FUNCTION_BLOCK encodeIOpCdt (* CAT Function Block Type *)
  (* Standard: 61499-2 *)
  (* Version 0.0, 6/7/2026, Schneider Electric, template *)
  PACKAGE SE.Nereda;
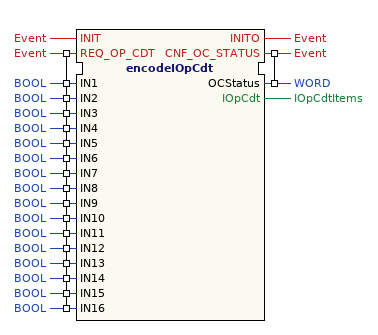
  EVENT_INPUT
    INIT;
    REQ_OP_CDT WITH IN1, IN2, IN3, IN4, IN5, IN6, IN7, IN8, IN9, IN10, IN11, IN12, IN13, IN14, IN15, IN16; (* Normal Execution Request *)
  END_EVENT
  EVENT_OUTPUT
    INITO;
    CNF_OC_STATUS WITH OCStatus; (* Execution Confirmation *)
  END_EVENT
  VAR_INPUT
    IN1 : BOOL; (* Argument *)
    IN2 : BOOL; (* Argument *)
    IN3 : BOOL; (* Argument *)
    IN4 : BOOL; (* Argument *)
    IN5 : BOOL; (* Argument *)
    IN6 : BOOL; (* Argument *)
    IN7 : BOOL; (* Argument *)
    IN8 : BOOL; (* Argument *)
    IN9 : BOOL; (* Argument *)
    IN10 : BOOL; (* Argument *)
    IN11 : BOOL; (* Argument *)
    IN12 : BOOL; (* Argument *)
    IN13 : BOOL; (* Argument *)
    IN14 : BOOL; (* Argument *)
    IN15 : BOOL; (* Argument *)
    IN16 : BOOL; (* Argument *)
  END_VAR
  VAR_OUTPUT
    OCStatus : WORD; (* Output bit image, bit 0 is the LSB of OUT1 *)
  END_VAR
  PLUGS
    IOpCdt : IOpCdtItems;
  END_PLUGS
  (* 01 - FUNCTIONNAL INPUT INTERFACE *)
  (* 05 - LOGIC *)
  (* 02 - FUNCTIONNAL OUTPUT INTERFACE *)
  (* 00 - INITIALIZATION *)
  (* 06 - HMI INTERFACE *)
  (* 03 - FIELD INTERFACE *)
  FBS
    OpCdts : AND_173860434676319F4; {SET_ATTRIBUTE(Configuration.GenericFBType.InterfaceParams, Runtime.Standard#CNT:=16;OUT:BOOL)}
    encodeB1 : VALFORMAT_95B1C22C7F49B890(FORMAT := '%s%s%s%s'); {SET_ATTRIBUTE(Configuration.GenericFBType.InterfaceParams, Runtime.Standard#I:=4;VALUE${I$}:INT,INT,INT,INT)}
    encodeB2 : VALFORMAT_95B1C22C7F49B890(FORMAT := '%s%s%s%s'); {SET_ATTRIBUTE(Configuration.GenericFBType.InterfaceParams, Runtime.Standard#I:=4;VALUE${I$}:INT,INT,INT,INT)}
    OpCdtsSmooth : boolValueChanged;
    encodeB3 : VALFORMAT_95B1C22C7F49B890(FORMAT := '%s%s%s%s'); {SET_ATTRIBUTE(Configuration.GenericFBType.InterfaceParams, Runtime.Standard#I:=4;VALUE${I$}:INT,INT,INT,INT)}
    encodeB4 : VALFORMAT_95B1C22C7F49B890(FORMAT := '%s%s%s%s'); {SET_ATTRIBUTE(Configuration.GenericFBType.InterfaceParams, Runtime.Standard#I:=4;VALUE${I$}:INT,INT,INT,INT)}
    IThis : encodeIOpCdt_HMI(QI := TRUE);
    OC_StatusWordConvert : BITMAN_182F748F2FAD4D59; {SET_ATTRIBUTE(Configuration.GenericFBType.InterfaceParams, Runtime.Standard#CNTIN:=16;CNTOUT:=1;IN${CNTIN$}:BOOL,BOOL,BOOL,BOOL,BOOL,BOOL,BOOL,BOOL,BOOL,BOOL,BOOL,BOOL,BOOL,BOOL,BOOL,BOOL;OUT${CNTOUT$}:WORD)}
    NOT_INs : NOT_21661D42DA8232174; {SET_ATTRIBUTE(Configuration.GenericFBType.InterfaceParams, Runtime.Standard#CNT:=16;OUT${CNT$}:BOOL,BOOL,BOOL,BOOL,BOOL,BOOL,BOOL,BOOL,BOOL,BOOL,BOOL,BOOL,BOOL,BOOL,BOOL,BOOL)}
    STR2INT1 : STR2INT;
    STR2INT2 : STR2INT;
    STR2INT3 : STR2INT;
    STR2INT4 : STR2INT;
    BOOL2INT1 : BOOL2INT_4;
    BOOL2INT2 : BOOL2INT_4;
    BOOL2INT3 : BOOL2INT_4;
    BOOL2INT4 : BOOL2INT_4;
    MemoOCStatus : MemoOC;
    StatusSmooth : WordValueChanged;
  END_FBS
  EVENT_CONNECTIONS
    REQ_OP_CDT TO OpCdts.REQ;
    OpCdts.CNF TO OpCdtsSmooth.REQ;
    OC_StatusWordConvert.INITO TO INITO;
    NOT_INs.CNF TO OC_StatusWordConvert.REQ;
    StatusSmooth.350834820611931F TO CNF_OC_STATUS;
    BOOL2INT1.6FC99A5BD1C38561 TO encodeB1.REQ;
    encodeB1.CNF TO STR2INT1.DD5870AA881150BB;
    BOOL2INT2.6FC99A5BD1C38561 TO encodeB2.REQ;
    encodeB2.CNF TO STR2INT2.DD5870AA881150BB;
    STR2INT1.6FC99A5BD1C38561 TO BOOL2INT2.DD5870AA881150BB;
    BOOL2INT3.6FC99A5BD1C38561 TO encodeB3.REQ;
    encodeB3.CNF TO STR2INT3.DD5870AA881150BB;
    BOOL2INT4.6FC99A5BD1C38561 TO encodeB4.REQ;
    encodeB4.CNF TO STR2INT4.DD5870AA881150BB;
    OpCdtsSmooth.CNF TO BOOL2INT1.DD5870AA881150BB;
    STR2INT2.6FC99A5BD1C38561 TO BOOL2INT3.DD5870AA881150BB;
    STR2INT3.6FC99A5BD1C38561 TO BOOL2INT4.DD5870AA881150BB;
    STR2INT4.6FC99A5BD1C38561 TO NOT_INs.REQ;
    StatusSmooth.350834820611931F TO IOpCdt.0DE1D11A791E8338;
    OpCdtsSmooth.CHD TO IOpCdt.51FD4CCF54DA16B0;
    OC_StatusWordConvert.CNF TO StatusSmooth.77F8F9CFF707DAFF;
    StatusSmooth.93AE3729A9342678 TO MemoOCStatus.7DC0949B91268FF6;
    INIT TO IThis.7D98611DC811A4F7;
    IThis.8A8403C8DB481D6C TO IThis.A665539B906F6DBA;
    MemoOCStatus.3B88FC64E51ED000 TO IThis.E03002787A644D63;
    IThis.8A8403C8DB481D6C TO OC_StatusWordConvert.INIT;
    IThis.6D29BCFC45D76FE3 TO IOpCdt.0DE1D11A791E8338;
    MemoOCStatus.3B88FC64E51ED000 TO IOpCdt.510B9224626AA5DB;
  END_CONNECTIONS
  DATA_CONNECTIONS
    IN1 TO OpCdts.IN1;
    IN2 TO OpCdts.IN2;
    IN16 TO OpCdts.IN16;
    IN15 TO OpCdts.IN15;
    IN14 TO OpCdts.IN14;
    IN13 TO OpCdts.IN13;
    IN12 TO OpCdts.IN12;
    IN11 TO OpCdts.IN11;
    IN10 TO OpCdts.IN10;
    IN9 TO OpCdts.IN9;
    IN8 TO OpCdts.IN8;
    IN7 TO OpCdts.IN7;
    IN6 TO OpCdts.IN6;
    IN5 TO OpCdts.IN5;
    IN4 TO OpCdts.IN4;
    IN3 TO OpCdts.IN3;
    OpCdts.OUT TO OpCdtsSmooth.Input;
    NOT_INs.OUT16 TO OC_StatusWordConvert.IN16;
    NOT_INs.OUT1 TO OC_StatusWordConvert.IN1;
    NOT_INs.OUT2 TO OC_StatusWordConvert.IN2;
    NOT_INs.OUT3 TO OC_StatusWordConvert.IN3;
    NOT_INs.OUT4 TO OC_StatusWordConvert.IN4;
    NOT_INs.OUT5 TO OC_StatusWordConvert.IN5;
    NOT_INs.OUT6 TO OC_StatusWordConvert.IN6;
    NOT_INs.OUT7 TO OC_StatusWordConvert.IN7;
    NOT_INs.OUT8 TO OC_StatusWordConvert.IN8;
    NOT_INs.OUT9 TO OC_StatusWordConvert.IN9;
    NOT_INs.OUT10 TO OC_StatusWordConvert.IN10;
    NOT_INs.OUT11 TO OC_StatusWordConvert.IN11;
    NOT_INs.OUT12 TO OC_StatusWordConvert.IN12;
    NOT_INs.OUT13 TO OC_StatusWordConvert.IN13;
    NOT_INs.OUT14 TO OC_StatusWordConvert.IN14;
    NOT_INs.OUT15 TO OC_StatusWordConvert.IN15;
    IN1 TO NOT_INs.IN1;
    IN2 TO NOT_INs.IN2;
    IN3 TO NOT_INs.IN3;
    IN4 TO NOT_INs.IN4;
    IN5 TO NOT_INs.IN5;
    IN6 TO NOT_INs.IN6;
    IN7 TO NOT_INs.IN7;
    IN8 TO NOT_INs.IN8;
    IN9 TO NOT_INs.IN9;
    IN10 TO NOT_INs.IN10;
    IN11 TO NOT_INs.IN11;
    IN12 TO NOT_INs.IN12;
    IN13 TO NOT_INs.IN13;
    IN14 TO NOT_INs.IN14;
    IN15 TO NOT_INs.IN15;
    IN16 TO NOT_INs.IN16;
    StatusSmooth.AA81B8787A42C5C8 TO OCStatus;
    encodeB1.RESULT TO STR2INT1.4573FC8F228EB71D;
    BOOL2INT1.A6DEF5F9C27C1848 TO encodeB1.VALUE1;
    BOOL2INT1.515A2E3BB78F58C7 TO encodeB1.VALUE2;
    BOOL2INT1.FCA64FB4B13F606F TO encodeB1.VALUE3;
    BOOL2INT1.740A810221DABFBE TO encodeB1.VALUE4;
    BOOL2INT2.A6DEF5F9C27C1848 TO encodeB2.VALUE1;
    BOOL2INT2.515A2E3BB78F58C7 TO encodeB2.VALUE2;
    BOOL2INT2.FCA64FB4B13F606F TO encodeB2.VALUE3;
    BOOL2INT2.740A810221DABFBE TO encodeB2.VALUE4;
    encodeB2.RESULT TO STR2INT2.4573FC8F228EB71D;
    BOOL2INT3.A6DEF5F9C27C1848 TO encodeB3.VALUE1;
    BOOL2INT3.515A2E3BB78F58C7 TO encodeB3.VALUE2;
    BOOL2INT3.FCA64FB4B13F606F TO encodeB3.VALUE3;
    BOOL2INT3.740A810221DABFBE TO encodeB3.VALUE4;
    encodeB3.RESULT TO STR2INT3.4573FC8F228EB71D;
    BOOL2INT4.A6DEF5F9C27C1848 TO encodeB4.VALUE1;
    BOOL2INT4.515A2E3BB78F58C7 TO encodeB4.VALUE2;
    BOOL2INT4.FCA64FB4B13F606F TO encodeB4.VALUE3;
    BOOL2INT4.740A810221DABFBE TO encodeB4.VALUE4;
    encodeB4.RESULT TO STR2INT4.4573FC8F228EB71D;
    IN4 TO BOOL2INT1.4573FC8F228EB71D;
    IN3 TO BOOL2INT1.DF8224FEB3446E92;
    IN2 TO BOOL2INT1.F547CEFAFDE5D422;
    IN1 TO BOOL2INT1.25941BC08BA9FF7D;
    IN8 TO BOOL2INT2.4573FC8F228EB71D;
    IN7 TO BOOL2INT2.DF8224FEB3446E92;
    IN6 TO BOOL2INT2.F547CEFAFDE5D422;
    IN5 TO BOOL2INT2.25941BC08BA9FF7D;
    IN12 TO BOOL2INT3.4573FC8F228EB71D;
    IN11 TO BOOL2INT3.DF8224FEB3446E92;
    IN10 TO BOOL2INT3.F547CEFAFDE5D422;
    IN9 TO BOOL2INT3.25941BC08BA9FF7D;
    IN16 TO BOOL2INT4.4573FC8F228EB71D;
    IN15 TO BOOL2INT4.DF8224FEB3446E92;
    IN14 TO BOOL2INT4.F547CEFAFDE5D422;
    IN13 TO BOOL2INT4.25941BC08BA9FF7D;
    OpCdtsSmooth.Output TO IOpCdt.5E924D1CC4B831CF;
    STR2INT1.A6DEF5F9C27C1848 TO IOpCdt.87CAB742E188E408;
    STR2INT2.A6DEF5F9C27C1848 TO IOpCdt.315583C88EDCE2AB;
    STR2INT3.A6DEF5F9C27C1848 TO IOpCdt.DC6E7346CAD3F412;
    STR2INT4.A6DEF5F9C27C1848 TO IOpCdt.154499D847362610;
    OC_StatusWordConvert.OUT1 TO StatusSmooth.25B5287A5784F3EC;
    StatusSmooth.AA81B8787A42C5C8 TO MemoOCStatus.B48D4147D400E339;
    IThis.74E1E0951D70046E TO IOpCdt.83A3C315F80CFE17;
    IThis.EE9470BA0350B131 TO IOpCdt.B50BFE7459784F00;
    IThis.EDAEBE4CEBDB9AE9 TO IOpCdt.946A0F582B551978;
    IThis.521EB392A39EAFAC TO IOpCdt.FCEA282DF5077920;
    IThis.882EBDE88CE34770 TO IOpCdt.2B4F39E9175B3855;
    IThis.CFFC3D70D2D95759 TO IOpCdt.4596A1B27C10C2CD;
    IThis.FEED97F6C5CA5C81 TO IOpCdt.A9753615DA8DD82A;
    IThis.7E2A6F1CECD5D852 TO IOpCdt.824CE9000F3F9466;
    IThis.16A171A2C76E95DE TO IOpCdt.72067FEC91126715;
    IThis.7C8621FA46B2D015 TO IOpCdt.37C7DD09745BE300;
    IThis.16CDB416492184BE TO IOpCdt.03CAF86670282F7A;
    IThis.852B9ADF3B1DF3DB TO IOpCdt.A578CCE6834280A9;
    IThis.779E1C38D576D599 TO IOpCdt.932E293892006A0F;
    IThis.80EDC56ADCA55E5B TO IOpCdt.3136228301C0A3F6;
    IThis.FA6EA3B49E681876 TO IOpCdt.BBA5573FBFE93EF1;
    IThis.C7252B37E7A4B5F2 TO IOpCdt.9095F08A1259C467;
    MemoOCStatus.7D0D48F0603D0B5F TO IThis.874756052129F02D;
    MemoOCStatus.3633FC608AFD6DED TO IThis.4BC035DD1E74A476;
    MemoOCStatus.7BB35991AF3AC8C5 TO IThis.4B2762FA5AEA2C62;
    MemoOCStatus.4002808179853F91 TO IThis.A0359A9DEE65770A;
    MemoOCStatus.4B917ED4557C577F TO IThis.AF79EA3753C9604B;
    MemoOCStatus.6E2561F6A492C21C TO IThis.B7A123C4DFD74089;
    MemoOCStatus.40632A3525912577 TO IThis.0DF76C0E5E990D90;
    MemoOCStatus.51E24AFC21EC80FD TO IThis.93107A7AF8A3FD05;
    MemoOCStatus.4E31ABC595FC99C5 TO IThis.17859EFEEE340DD7;
    MemoOCStatus.7340464A92B25B83 TO IThis.443273E361A83C2E;
    MemoOCStatus.7F58593D76CC17D5 TO IOpCdt.7FD7CF3BAAB2C8B1;
  END_CONNECTIONS
END_FUNCTION_BLOCK
